{attribute 'enable_dynamic_creation'}
FUNCTION_BLOCK Circle EXTENDS Disposable IMPLEMENTS I_DrawableShape
VAR
	_radius: INT;
END_VAR

METHOD Clone : I_DrawableShape
VAR
	pCircle : POINTER TO Circle;	
END_VAR
pCircle := __NEW(Circle);
pCircle^.radius := radius;
Clone := pCircle^;
END_METHOD


METHOD Draw

VAR
	str : STRING;
END_VAR
str := TO_STRING(radius);
ADSLOGSTR(msgCtrlMask :=ADSLOG_MSGTYPE_HINT, msgFmtStr :='Draw circle with radius: %s', strArg := str);
END_METHOD

PROPERTY Radius : INT
GET
Radius := _radius;
END_GET
SET
_radius := Radius;
END_SET
END_PROPERTY

END_FUNCTION_BLOCK

(* stored: Version 1.1.0.1, ProductVersion 3.1.4024.12
   POU Circle: Id {7bf41376-fe79-4fc9-9b0f-cc0bfa7817da}, SpecialFunc None
   Method Clone: Id {40bc29e0-bf78-4d5d-8f5d-1f786394c013}
   Method Draw: Id {919be77b-1433-43bb-9e6d-ebea1c177f82}
   Property Radius: Id {a34de360-bafa-47b2-9b5a-87523dbf7965}
   Get Get: Id {b4b1e14d-2cb6-4d31-9d39-7bdd833041a6}
   Set Set: Id {ad4d0cb0-75ea-4310-9847-518237d41bcb} *)
